// TIA Portal V21 export
FUNCTION "GestProfinetAbilitazionedispositivo" : Void   // FC100, LAD
{ S7_Optimized_Access := 'TRUE' }
// stored: SetENOAutomatically false
BEGIN

REGION Network 1 (SCL)
   // D_ACT_DP(REQ:=_bool_in_, MODE:=_usint_in_, LADDR:=_hw_any_in_, BUSY=>_bool_out_)
END_REGION
END_FUNCTION
